Staubli VAL3: VelocityCfgMsg.dtx

public Prefix prefix
  [0]
    num nLength
    num nData[4]
public Header header
  [0]
    num nMsgType
    num nCommType
    num nReplyCode
    num nData[12]
public Body body
  [0]
    num nData[68]
public VelocityCfg velCfg
  [0]
    num nCmdType
    num nRefFrameVec[6]
    num nToolVec[6]
    num nAccel
    num nVel
    num nTransVel
    num nRotVel
